# EPICS IOC start-up script: iocsh/ethercatmcDefPos.iocsh
dbLoadRecords("ethercatmcDefPos.template", "P=$(P), R=$(R), MOTOR_PORT=$(MOTOR_PORT), ASYN_PORT=$(ASYN_PORT), AXIS_NO=$(AXIS_NO), PREC=$(PREC), EGU=$(EGU),NVL=$(NVL) ")
